// TIA Portal V20 export
FUNCTION_BLOCK "AdjScanner"   // FB510, FBD
{ S7_Optimized_Access := 'TRUE' }
// stored: AutoNumber false, MemoryReserve 100, SetENOAutomatically false
   VAR
      Var { ExternalAccessible := 'False'; ExternalVisible := 'False'; ExternalWritable := 'False'} : "TypeVar";
      Cmd { ExternalAccessible := 'False'; ExternalVisible := 'False'; ExternalWritable := 'False'} : "TypeCmd";
      SIO { ExternalAccessible := 'False'; ExternalVisible := 'False'; ExternalWritable := 'False'} : "SysBaluffBUS007F";
      Pos { ExternalAccessible := 'False'; ExternalVisible := 'False'; ExternalWritable := 'False'} : "SysPos";
      "M" { ExternalAccessible := 'False'; ExternalVisible := 'False'; ExternalWritable := 'False'} : "SysMotor";
      TAreaOn { ExternalAccessible := 'False'; ExternalVisible := 'False'; ExternalWritable := 'False'} : TON_TIME;
      TAutoOn { ExternalAccessible := 'False'; ExternalVisible := 'False'; ExternalWritable := 'False'} : TON_TIME;
      TAutoTarPosManOn { ExternalAccessible := 'False'; ExternalVisible := 'False'; ExternalWritable := 'False'} : TON_TIME;
      TPosRestart { ExternalAccessible := 'False'; ExternalVisible := 'False'; ExternalWritable := 'False'} : TON_TIME;
      tarOld { ExternalAccessible := 'False'; ExternalVisible := 'False'; ExternalWritable := 'False'} : DInt;
      autoTarPosMan { ExternalAccessible := 'False'; ExternalVisible := 'False'; ExternalWritable := 'False'} : Bool;
      refTarPos { ExternalAccessible := 'False'; ExternalVisible := 'False'; ExternalWritable := 'False'} : DInt;
      posRestart { ExternalAccessible := 'False'; ExternalVisible := 'False'; ExternalWritable := 'False'} : Bool;
      posOk { ExternalAccessible := 'False'; ExternalVisible := 'False'; ExternalWritable := 'False'} : Bool;
      posRegActive { ExternalAccessible := 'False'; ExternalVisible := 'False'; ExternalWritable := 'False'} : Bool;
   END_VAR
   VAR_TEMP
      CtrlPc : Struct
         ackErr : Bool;
         manModeActive : Bool;
         manP : Bool;
         manM : Bool;
         manRefRun : Bool;
      END_STRUCT;
      refPosDiff : DInt;
      areaDelayOn : Bool;
      offsetZeroPoint : Real;
      TarTolMin : Real;
      TarTolMax : Real;
      PosOkTolMin : Real;
      PosOkTolMax : Real;
      tolerance : Real;
      regPoint : Real;
   END_VAR
BEGIN

REGION Network 1 (SCL): calibration value from pc
   "ComSd".Data.Scanner.SetCalibratePosOk := FALSE;

   IF "ComRd".Data.Scanner.SetCalibratePos THEN

       IF "G".Cfg.modeBoardPassing = 3 THEN
           "Enc"."8B1.B".refPos := 0;
       ELSIF "G".Cfg.modeBoardPassing = 2 THEN
           "Enc"."8B1.B".refPos := (DINT_TO_REAL("ComRd".Data.Scanner.TargetPos) / 10.0) * -1.0;
       ELSE
           "Enc"."8B1.B".refPos := DINT_TO_REAL("ComRd".Data.Scanner.TargetPos) / 10.0;
       END_IF;
       "ComSd".Data.Scanner.SetCalibratePosOk := TRUE;
       "Enc"."8B1.B".ref := TRUE;
   END_IF;
END_REGION

REGION Network 2 (SCL): standardisation batch
   (* 
   if standardisation batch is active then the scanner status display should be off
   *)
   IF "ComRd".Data.Scanner.CalibratePos = -1 THEN
       "G".Batch.stdActive := TRUE;
   ELSE
       "G".Batch.stdActive := FALSE;
   END_IF;
END_REGION

REGION Network 3 (SCL): offset scanner
   (* 
   used with left AND right alignement to avoid the problem that a
   camera cannot position because is in mecanical limit switch
   ex.: right camera cannot reach position because is on minimum limit switch,
   so we move the scanner with an offset of 20 mm  more to the right side
   *)
   "Enc"."8B1.B".offset := DINT_TO_REAL(LIMIT_DINT(MN := -50, IN := "ComRd".Data.Scanner.RefPosToBoard, MX := 50));
END_REGION

REGION Network 4 (SCL): target position
   IF "G".comOk THEN
       #Cmd.target := DINT_TO_REAL("ComRd".Data.Scanner.TargetPos) / 10.0;
   END_IF;

   IF "G".Cfg.modeBoardPassing = 3 THEN
       #Cmd.target := 0.0;
   END_IF;

   IF #autoTarPosMan THEN
       #Cmd.target := DINT_TO_REAL("ComRd".Data.Scanner.TargetPos) / 10.0;
   END_IF;

   IF "G".Cfg.modeBoardPassing = 2 THEN
       #Cmd.target := #Cmd.target * -1.0 ;
   END_IF;

   "Ref".adjScannerTar :=  #Cmd.target + "Enc"."8B1.B".offset;
END_REGION

REGION Network 5 (SCL): data from pc
   IF NOT "G".errComPc THEN
       #CtrlPc.manModeActive := "ComRd".Data.Scanner.ManModeActive;
       #CtrlPc.manRefRun := "ComRd".Data.Scanner.ManRefRun;
       IF "G".Cfg.modeBoardPassing = 2 THEN
           #CtrlPc.manP := "ComRd".Data.Scanner.ManMinus;
           #CtrlPc.manM := "ComRd".Data.Scanner.ManPlus;
       ELSE
           #CtrlPc.manP := "ComRd".Data.Scanner.ManPlus;
           #CtrlPc.manM := "ComRd".Data.Scanner.ManMinus;
       END_IF;
   ELSE
       #CtrlPc.manModeActive := TRUE;
       #CtrlPc.manP := FALSE;
       #CtrlPc.manM := FALSE;
       #CtrlPc.manRefRun := FALSE;
   END_IF;
   #CtrlPc.ackErr := "G".ack;
END_REGION

REGION Network 6: off
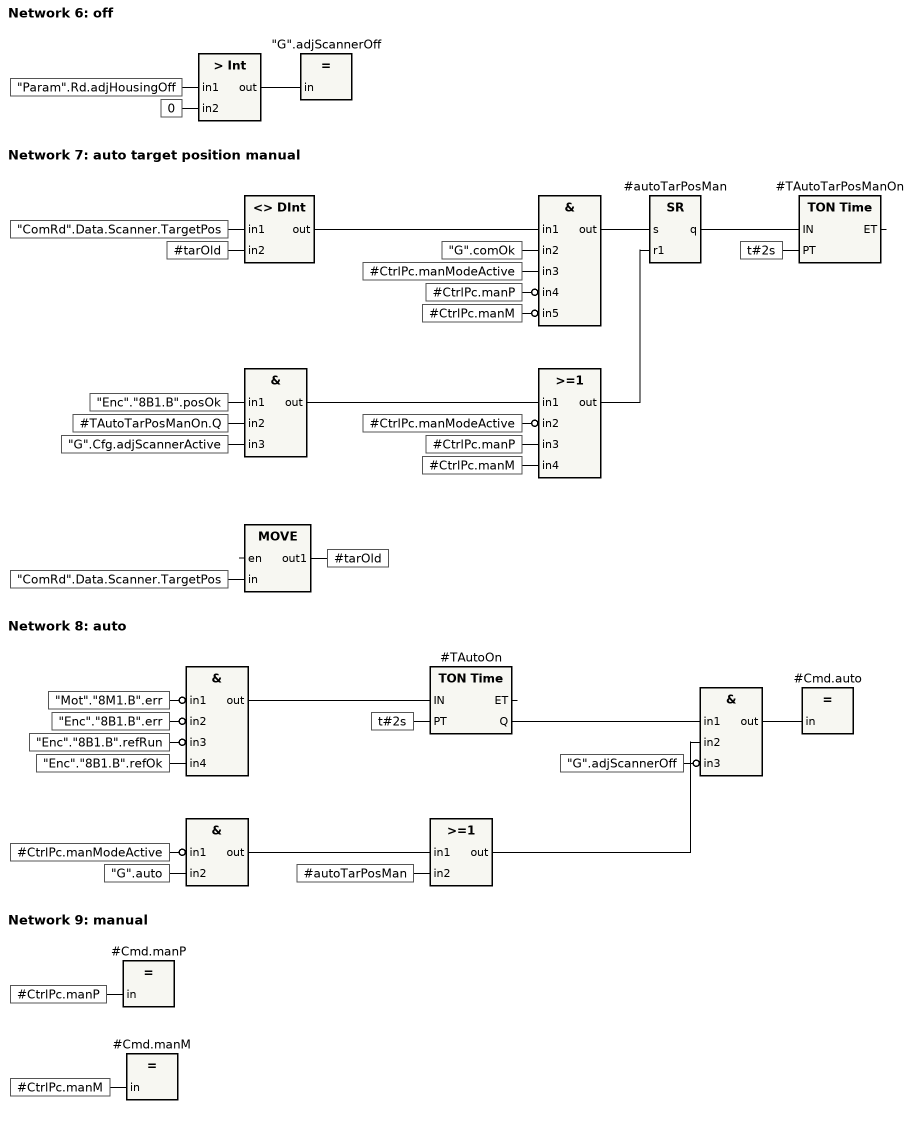
   "G".adjScannerOff := "Param".Rd.adjHousingOff > 0;
END_REGION

REGION Network 7: auto target position manual
   IF ("ComRd".Data.Scanner.TargetPos <> #tarOld) AND "G".comOk AND #CtrlPc.manModeActive AND NOT #CtrlPc.manP AND NOT #CtrlPc.manM THEN
       #autoTarPosMan := TRUE;   // SR flip-flop
   END_IF;
   IF ("Enc"."8B1.B".posOk AND #TAutoTarPosManOn.Q AND "G".Cfg.adjScannerActive) OR NOT #CtrlPc.manModeActive OR #CtrlPc.manP OR #CtrlPc.manM THEN
       #autoTarPosMan := FALSE;
   END_IF;
   #TAutoTarPosManOn(IN := #autoTarPosMan, PT := t#2s);   // TON
   #tarOld := "ComRd".Data.Scanner.TargetPos;
END_REGION

REGION Network 8: auto
   #TAutoOn(IN := NOT "Mot"."8M1.B".err AND NOT "Enc"."8B1.B".err AND NOT "Enc"."8B1.B".refRun AND "Enc"."8B1.B".refOk,   // TON
            PT := t#2s);
   #Cmd.auto := #TAutoOn.Q AND ((NOT #CtrlPc.manModeActive AND "G".auto) OR #autoTarPosMan) AND NOT "G".adjScannerOff;
END_REGION

REGION Network 9: manual
   #Cmd.manP := #CtrlPc.manP;
   #Cmd.manM := #CtrlPc.manM;
END_REGION

REGION Network 10 (SCL): calibration value
   "Enc"."8B1.B".calGain := 0.1;

   "Enc"."8B1.B".minPos := -500.0;
   "Enc"."8B1.B".maxPos := 500.0;

   "Enc"."8B1.B".limMin := "Enc"."8B1.B".minPos - 5.0;
   "Enc"."8B1.B".limMax := "Enc"."8B1.B".maxPos + 5.0;

   "Enc"."8B1.B".tarMinPos := "Enc"."8B1.B".minPos + 0.0;
   "Enc"."8B1.B".tarMaxPos := "Enc"."8B1.B".maxPos - 0.0;

   #offsetZeroPoint := -117.3;
END_REGION

REGION Network 12: sensor IO-Link adjustment scannerhousing
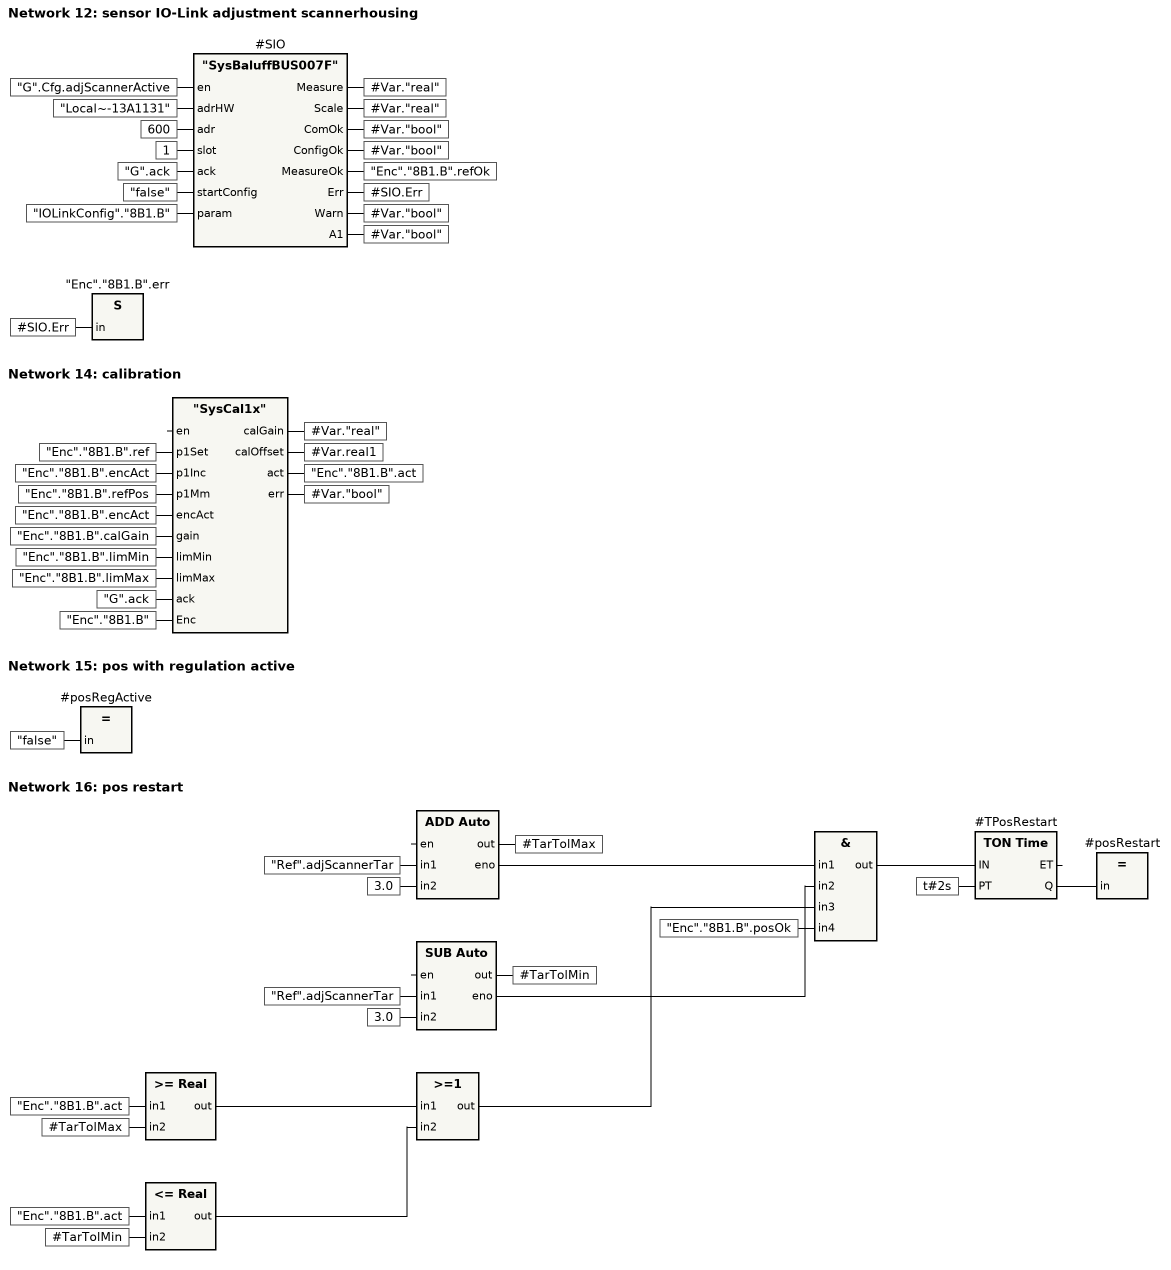
   IF "G".Cfg.adjScannerActive THEN
       #SIO(adrHW := "Local~-13A1131",   // "SysBaluffBUS007F"
            adr := 600,
            slot := 1,
            ack := "G".ack,
            startConfig := "false",
            param := "IOLinkConfig"."8B1.B",
            Measure => #Var."real",
            Scale => #Var."real",
            ComOk => #Var."bool",
            ConfigOk => #Var."bool",
            MeasureOk => "Enc"."8B1.B".refOk,
            Err => #SIO.Err,
            Warn => #Var."bool",
            A1 => #Var."bool");
   END_IF;
   IF #SIO.Err THEN "Enc"."8B1.B".err := TRUE; END_IF;
END_REGION

REGION Network 13 (SCL): sensor IO-Link adjustment scannerhousing - copy data
   "Enc"."8B1.B".encAct := REAL_TO_DINT((#SIO.Measure + #offsetZeroPoint) * 10.0);
END_REGION

REGION Network 14: calibration
   "SysCal1x"(p1Set := "Enc"."8B1.B".ref,
              p1Inc := "Enc"."8B1.B".encAct,
              p1Mm := "Enc"."8B1.B".refPos,
              encAct := "Enc"."8B1.B".encAct,
              gain := "Enc"."8B1.B".calGain,
              limMin := "Enc"."8B1.B".limMin,
              limMax := "Enc"."8B1.B".limMax,
              ack := "G".ack,
              Enc := "Enc"."8B1.B",
              calGain => #Var."real",
              calOffset => #Var.real1,
              act => "Enc"."8B1.B".act,
              err => #Var."bool");
END_REGION

REGION Network 15: pos with regulation active
   #posRegActive := "false";
END_REGION

REGION Network 16: pos restart
   #TarTolMax := "Ref".adjScannerTar + 3.0;
   #TarTolMin := "Ref".adjScannerTar - 3.0;
   #TPosRestart(IN := (("Enc"."8B1.B".act >= #TarTolMax) OR ("Enc"."8B1.B".act <= #TarTolMin)) AND "Enc"."8B1.B".posOk,   // TON
                PT := t#2s);
   #posRestart := #TPosRestart.Q;
END_REGION

REGION Network 17: pos param
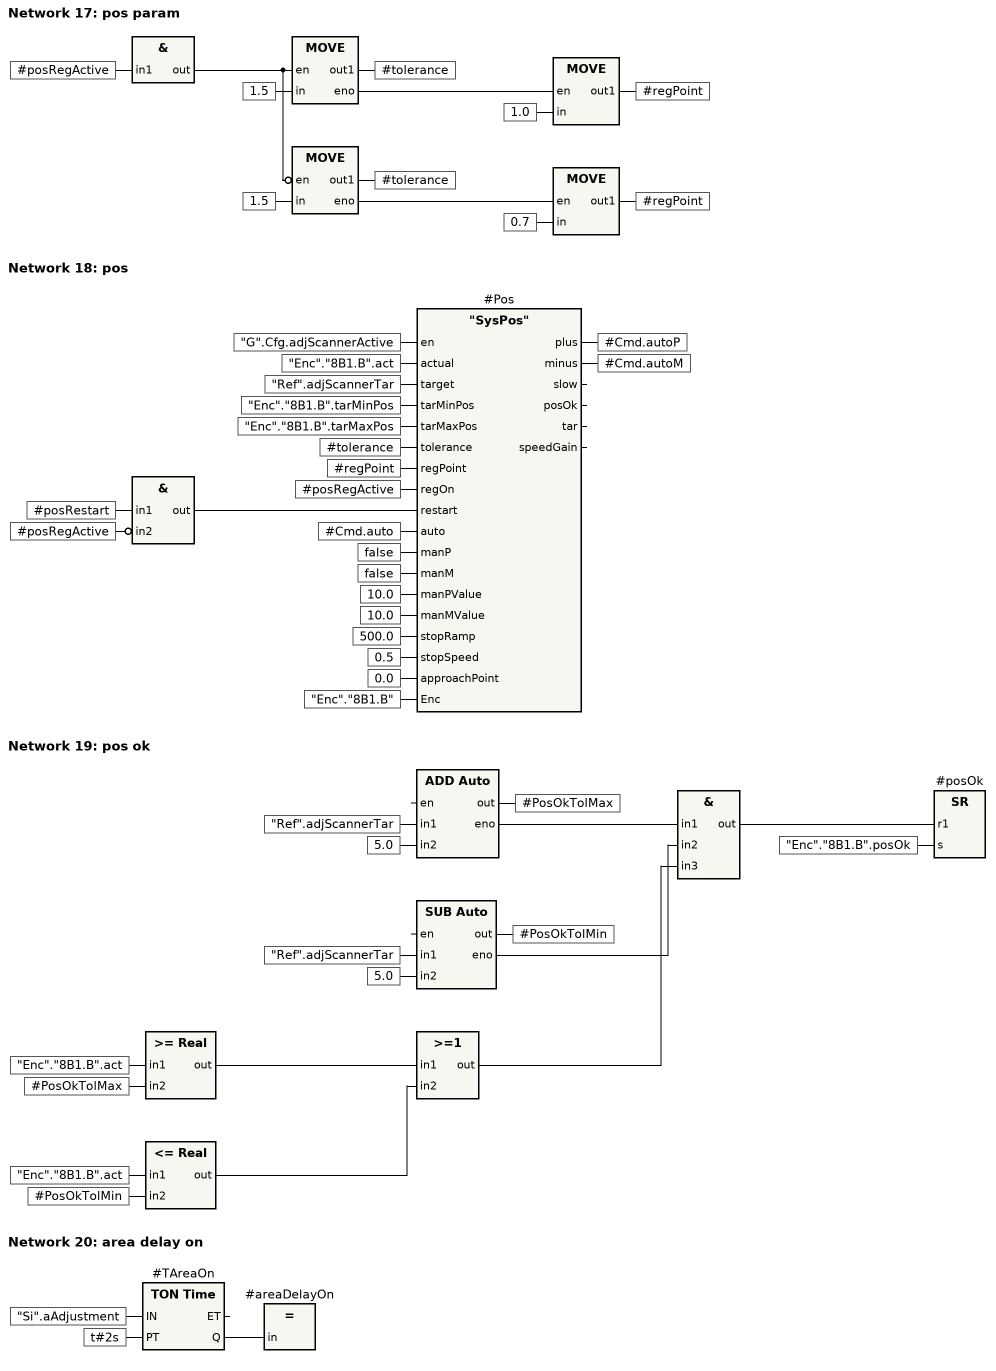
   IF #posRegActive THEN
       #tolerance := 1.5;
       #regPoint := 1.0;
   END_IF;
   IF NOT #posRegActive THEN
       #tolerance := 1.5;
       #regPoint := 0.7;
   END_IF;
END_REGION

REGION Network 18: pos
   IF "G".Cfg.adjScannerActive THEN
       #Pos(actual := "Enc"."8B1.B".act,   // "SysPos"
            target := "Ref".adjScannerTar,
            tarMinPos := "Enc"."8B1.B".tarMinPos,
            tarMaxPos := "Enc"."8B1.B".tarMaxPos,
            tolerance := #tolerance,
            regPoint := #regPoint,
            regOn := #posRegActive,
            restart := #posRestart AND NOT #posRegActive,
            auto := #Cmd.auto,
            manP := false,
            manM := false,
            manPValue := 10.0,
            manMValue := 10.0,
            stopRamp := 500.0,
            stopSpeed := 0.5,
            approachPoint := 0.0,
            Enc := "Enc"."8B1.B",
            plus => #Cmd.autoP,
            minus => #Cmd.autoM);
   END_IF;
END_REGION

REGION Network 19: pos ok
   #PosOkTolMax := "Ref".adjScannerTar + 5.0;
   #PosOkTolMin := "Ref".adjScannerTar - 5.0;
   IF "Enc"."8B1.B".posOk THEN
       #posOk := TRUE;   // SR flip-flop
   END_IF;
   IF ("Enc"."8B1.B".act >= #PosOkTolMax) OR ("Enc"."8B1.B".act <= #PosOkTolMin) THEN
       #posOk := FALSE;
   END_IF;
END_REGION

REGION Network 20: area delay on
   #TAreaOn(IN := "Si".aAdjustment, PT := t#2s);   // TON
   #areaDelayOn := #TAreaOn.Q;
END_REGION

REGION Network 21: motor
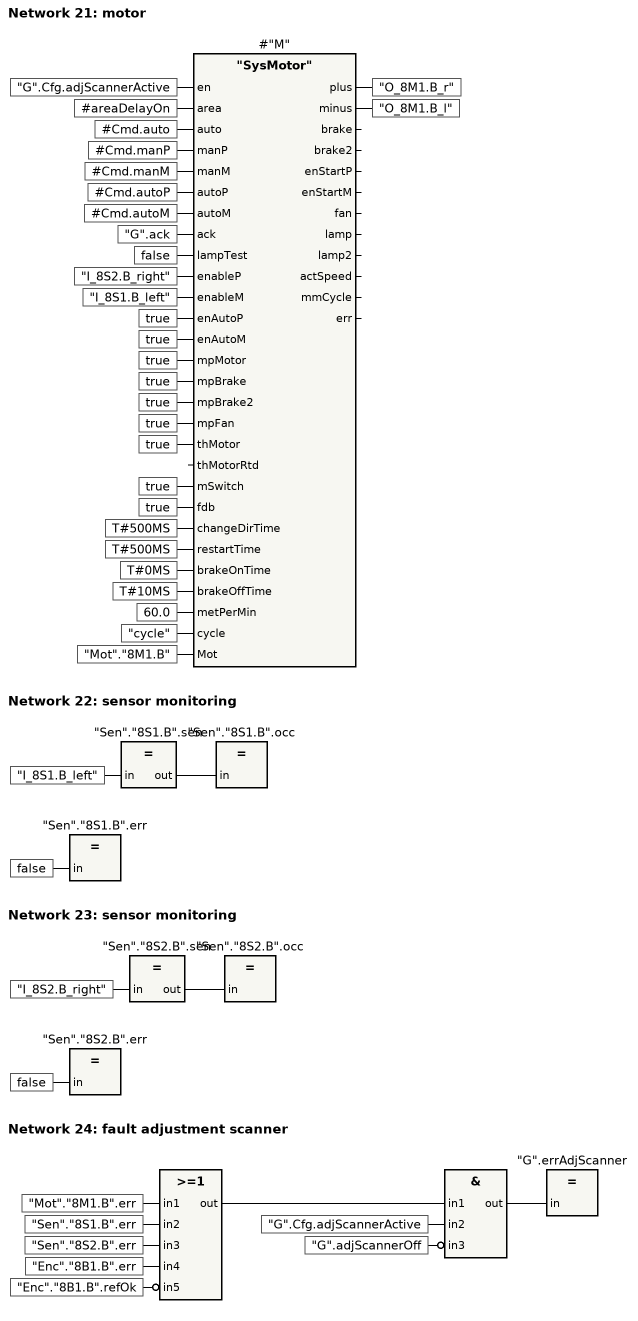
   IF "G".Cfg.adjScannerActive THEN
       #"M"(area := #areaDelayOn,   // "SysMotor"
            auto := #Cmd.auto,
            manP := #Cmd.manP,
            manM := #Cmd.manM,
            autoP := #Cmd.autoP,
            autoM := #Cmd.autoM,
            ack := "G".ack,
            lampTest := false,
            enableP := "I_8S2.B_right",
            enableM := "I_8S1.B_left",
            enAutoP := true,
            enAutoM := true,
            mpMotor := true,
            mpBrake := true,
            mpBrake2 := true,
            mpFan := true,
            thMotor := true,
            mSwitch := true,
            fdb := true,
            changeDirTime := T#500MS,
            restartTime := T#500MS,
            brakeOnTime := T#0MS,
            brakeOffTime := T#10MS,
            metPerMin := 60.0,
            cycle := "cycle",
            Mot := "Mot"."8M1.B",
            plus => "O_8M1.B_r",
            minus => "O_8M1.B_l");
   END_IF;
END_REGION

REGION Network 22: sensor monitoring
   "Sen"."8S1.B".sen := "I_8S1.B_left";
   "Sen"."8S1.B".occ := "I_8S1.B_left";
   "Sen"."8S1.B".err := false;
END_REGION

REGION Network 23: sensor monitoring
   "Sen"."8S2.B".sen := "I_8S2.B_right";
   "Sen"."8S2.B".occ := "I_8S2.B_right";
   "Sen"."8S2.B".err := false;
END_REGION

REGION Network 24: fault adjustment scanner
   "G".errAdjScanner := ("Mot"."8M1.B".err OR "Sen"."8S1.B".err OR "Sen"."8S2.B".err OR "Enc"."8B1.B".err OR NOT "Enc"."8B1.B".refOk) AND "G".Cfg.adjScannerActive AND NOT "G".adjScannerOff;
END_REGION

REGION Network 25 (SCL): data to pc
   IF "G".Cfg.adjScannerActive THEN
       "Ref".adjScannerAct := REAL_TO_DINT("Enc"."8B1.B".act * 10.0);
       "ComSd".Data.Scanner.ActualEncPos := "Enc"."8B1.B".encAct;
       IF "G".Cfg.modeBoardPassing = 2 THEN
           "ComSd".Data.Scanner.ActualPos := "Ref".adjScannerAct * -1;
           "ComSd".Data.Scanner.Plus := "Mot"."8M1.B".minus;
           "ComSd".Data.Scanner.Minus := "Mot"."8M1.B".plus;
       ELSE
           "ComSd".Data.Scanner.ActualPos := "Ref".adjScannerAct;
           "ComSd".Data.Scanner.Plus := "Mot"."8M1.B".plus;
           "ComSd".Data.Scanner.Minus := "Mot"."8M1.B".minus;
       END_IF;
       "ComSd".Data.Scanner.LimitSwitchMin := "Sen"."8S1.B".sen;
       "ComSd".Data.Scanner.LimitSwitchMax := "Sen"."8S2.B".sen;
       "ComSd".Data.Scanner.Err := "Mot"."8M1.B".err;
       "ComSd".Data.Scanner.ErrEnc := "Enc"."8B1.B".err;
       "ComSd".Data.Scanner.PosOk := ("Enc"."8B1.B".posOk AND #posRegActive) OR (#posOk AND NOT #posRegActive);
       "ComSd".Data.Scanner.refRun := "Enc"."8B1.B".refRun;
       "ComSd".Data.Scanner.refOk := "Enc"."8B1.B".refOk;
   ELSE
       "ComSd".Data.Scanner.ActualEncPos := 0;
       "ComSd".Data.Scanner.ActualPos := 0;
       "ComSd".Data.Scanner.LimitSwitchMin := FALSE;
       "ComSd".Data.Scanner.LimitSwitchMax := FALSE;
       "ComSd".Data.Scanner.Err := FALSE;
       "ComSd".Data.Scanner.ErrEnc := FALSE;
       "ComSd".Data.Scanner.PosOk := TRUE;
       "ComSd".Data.Scanner.Plus := FALSE;
       "ComSd".Data.Scanner.Minus := FALSE;
       "ComSd".Data.Scanner.refRun := FALSE;
       "ComSd".Data.Scanner.refOk := TRUE;
   END_IF;
END_REGION
END_FUNCTION_BLOCK
